// TIA Portal V19 export
TYPE "UDT_DINFAULTS"
   STRUCT
      ctrl : Array[0..15] of Bool;   // External data (Primary fault data - alarm & plc ackn)
      status : Array[0..15] of Bool;   // External data (Secondary fault data - siren & hmi ackn)
   END_STRUCT;
   // // ctrl[0] : Alarm 0
   // // ctrl[1] : Alarm 1
   // // ctrl[2] : Alarm 2
   // // ctrl[3] : Alarm 3
   // // ctrl[4] : Alarm 4
   // // ctrl[5] : Alarm 5
   // // ctrl[6] : Alarm 6
   // // ctrl[7] : Alarm 7
   // // ctrl[8] : PLC Ackn 0
   // // ctrl[9] : PLC Ackn 1
   // // ctrl[10] : PLC Ackn 2
   // // ctrl[11] : PLC Ackn 3
   // // ctrl[12] : PLC Ackn 4
   // // ctrl[13] : PLC Ackn 5
   // // ctrl[14] : PLC Ackn 6
   // // ctrl[15] : PLC Ackn 7
   // // status[0] : Siren 0
   // // status[1] : Siren 1
   // // status[2] : Siren 2
   // // status[3] : Siren 3
   // // status[4] : Siren 4
   // // status[5] : Siren 5
   // // status[6] : Siren 6
   // // status[7] : Siren 7
   // // status[8] : HMI Ackn 0
   // // status[9] : HMI Ackn 1
   // // status[10] : HMI Ackn 2
   // // status[11] : HMI Ackn 3
   // // status[12] : HMI Ackn 4
   // // status[13] : HMI Ackn 5
   // // status[14] : HMI Ackn 6
   // // status[15] : HMI Ackn 7
END_TYPE
